// TIA Portal project "Progetto_Arduino_Rev2" (V15)

(* hardware
DEVICE "S7-1200 station_1"  S7-1200 Station
   slot 0: "Rack_0"  S7-1200 Rack  Rack  V1.0
   slot 1: "PLC_1"  CPU 1211C AC/DC/Rly  6ES7 211-1BE40-0XB0  V4.2
*)

// ===== PLC "PLC_1"  CPU 1211C AC/DC/Rly =====

VAR_GLOBAL   // PLC tag table "Default tag table"
   "clock" AT %I0.0 : Bool;   // hsc clock
   "gate" AT %I0.3 : Bool;   // hsc gate
   "out0" AT %Q0.0 : Bool;
   "out1" AT %Q0.1 : Bool;
   "out2" AT %Q0.2 : Bool;
   "out3" AT %Q0.3 : Bool;
   "distance" AT %MD1 : Real;
   "interrupt_count" AT %MD16 : DInt;   // Count number of falling edges of hsc gate
   "Act_dist2" AT %MD33 : DInt;   // Valore da passare ad arduino che permette di settare la distanza del motore
   "Enable_Set_dist2" AT %M9.0 : Bool;
   "Direction" AT %M0.1 : Bool;
END_VAR

VAR_GLOBAL CONSTANT   // PLC tag table "Default tag table"
   "clock_period" : Real := 0.000001;   // period clock (seconds)
   "sound_speed" : Real := 340.0;   // (m/s)
   "Enable_Set_dist" : Bool := true;
   "Act_dist" : Int := 3;
END_VAR

DATA_BLOCK "Data_block_1"   // DB2
{ S7_Optimized_Access := 'TRUE' }
VERSION : 0.1
   VAR
      HSC_1 : HSC_Count;
   END_VAR
BEGIN
   HSC_1.EnHSC := true;
END_DATA_BLOCK

// folder: System blocks/Program resources

DATA_BLOCK "IEC_Timer_0_DB"   // DB3
{ S7_Optimized_Access := 'TRUE' }
AUTHOR : Simatic
FAMILY : IEC
NAME : IEC_TMR
VERSION : 1.0
// stored: InstanceOfName IEC_TIMER
"IEC_TIMER"
BEGIN
END_DATA_BLOCK

// folder: (top level)

ORGANIZATION_BLOCK "Main"   // OB1, LAD, ProgramCycle
TITLE = "Main Program Sweep (Cycle)"
{ S7_Optimized_Access := 'TRUE' }
VERSION : 0.1
   VAR_INPUT
      Initial_Call : Bool;   // Initial call of this OB
      Remanence : Bool;   // =True, if remanent data are available
   END_VAR
BEGIN
END_ORGANIZATION_BLOCK

ORGANIZATION_BLOCK "Cyclic interrupt"   // OB30, LAD, CyclicInterrupt
{ S7_Optimized_Access := 'TRUE' }
VERSION : 0.1
   VAR_INPUT
      Initial_Call : Bool;   // Initial call of this OB
      Event_Count : Int;   // Events discarded
   END_VAR
BEGIN

REGION Network 1
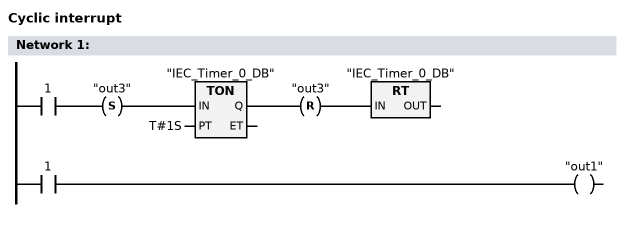
   // no checked SCL form for this network; see the picture
END_REGION
END_ORGANIZATION_BLOCK

ORGANIZATION_BLOCK "Hardware interrupt count"   // OB41, LAD, HWProcessInterrupt
{ S7_Optimized_Access := 'TRUE' }
VERSION : 0.1
   VAR_INPUT
      LADDR : Hw_Io;   // Hardware identifier
      USI : Word;   // User structure identifier
      IChannel : USInt;   // Interrupt channel number
      EventType : Byte;   // EventType
   END_VAR
BEGIN

REGION Network 1
   // Questo è i++
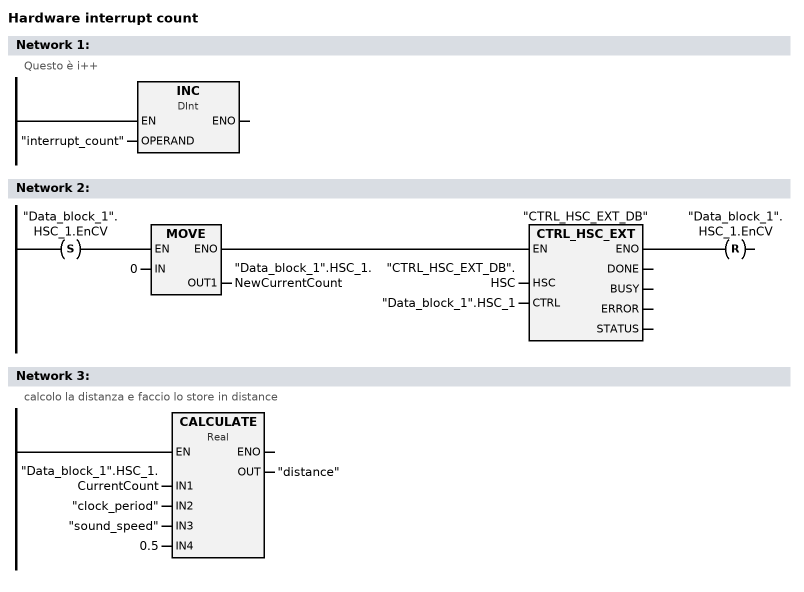
   RUNG wire#powerrail
      { S7_Templates := "DestType := DInt" } Inc( "interrupt_count" )
   END_RUNG
   // the same network as SCL:
   "interrupt_count" := "interrupt_count" + 1;
END_REGION

REGION Network 2
   // ENO of a box is taken as its EN; it also drops when the box reports an error
   "Data_block_1".HSC_1.EnCV := TRUE;
   "Data_block_1".HSC_1.NewCurrentCount := 0;
   "CTRL_HSC_EXT_DB"(HSC := "CTRL_HSC_EXT_DB".HSC, CTRL := "Data_block_1".HSC_1);   // CTRL_HSC_EXT
   "Data_block_1".HSC_1.EnCV := FALSE;
END_REGION

REGION Network 3
   // calcolo la distanza e faccio lo store in distance
   RUNG wire#powerrail
      { S7_Templates := "SrcType := Real"; S7_Expression := "IN1*IN2*IN3*IN4" } Calculate(in1 := "Data_block_1".HSC_1.CurrentCount, in2 := "clock_period", in3 := "sound_speed", in4 := 0.5, out => "distance")
   END_RUNG
   // the same network as SCL:
   "distance" := "Data_block_1".HSC_1.CurrentCount*"clock_period"*"sound_speed"*0.5;
END_REGION
END_ORGANIZATION_BLOCK